KUKA KRL program: Wood_Test.src, Wood_Test.dat

--- Wood_Test.src ---
&ACCESS RVEO
&REL 9
&PARAM DISKPATH = KRC:\R1\Program\Milling
DEF Wood_Test ( )
   INT lnActSt,lnUsedBase,lnUsedTool,lnBaseNr
   INT lnJobNr, lncounter, lncounter2
   FRAME lfZcut
   FRAME lfToolDiamShift
   FRAME lfStartMillingPos
   FRAME lfBaseShift
   FRAME lfBaseCycleZ

   CONTINUE
   ;IF ($T1 OR $T2)THEN
   GLOBAL INTERRUPT DECL 3 WHEN $STOPMESS==TRUE DO IR_STOPM ( )
   INTERRUPT ON 3
   BAS (#INITMOV,0)
   lnActSt = 1
   PTP $POS_ACT
;;ptp xhome
   ;ENDIF

   ; PTP XHOME
   SpindleRun(grUsedRPM,#CLOCKWISE)

   PTP lAstartPos

   ; Used Base and tool
   lnUsedBase = 11
   lnUsedTool = 11

   gnLastToolNr = 4
   lnBaseNr = 21

   gfMillingOffset = $NULLFRAME


   lfZcut = $NULLFRAME
   lfZcut.Z = 0
   lfBaseShift = {X 0,Y 0,Z 0,A 0,B 0,C 0}
   lfBaseCycleZ = $NULLFRAME
   lfBaseCycleZ.Z = 0

   ;*************************************************************
   ;*                      Mill TOP SURFACE                     *
   ;*************************************************************
   lfBaseCycleZ = $NULLFRAME
   lfBaseCycleZ.Z = 0
   BASE_DATA[lnUsedBase] = BASE_DATA[lnBaseNr] : lfBaseShift : lfBaseCycleZ
   TOOL_DATA[lnUsedTool] = TOOL_DATA[gnLastToolNr] :{X 0,Y 0,Z 0,A 270,B 0,C 0}

   MoveSettings(lnUsedBase, lnUsedTool, 100, grUsedMillingSpeed)
   ;; Move To PreposMillingPos Point P5 {5mm far from WP surface}
   lfToolDiamShift   = $NULLFRAME
   lfToolDiamShift.X = 0
   lfToolDiamShift.Y = grTool_Diameter[4]
   lfToolDiamShift.Z = 5
   lfStartMillingPos = lfWorkPos[5] : lfToolDiamShift
   LIN lfStartMillingPos

   ;; Move To Milling Point P5
   MoveSettings(lnUsedBase, lnUsedTool, 100, grUsedMillingSpeed)
   lfToolDiamShift   =   $NULLFRAME
   lfToolDiamShift.x =  0
   lfToolDiamShift.Y =  grTool_Diameter[4]
   lfToolDiamShift.Z =  0
   LIN lfWorkPos[5]:lfToolDiamShift C_VEL

   ;; Move To Milling Point P6
   MoveSettings(lnUsedBase, lnUsedTool, 100, grUsedMillingSpeed)
   lfToolDiamShift   =   $NULLFRAME
   lfToolDiamShift.x =  0
   lfToolDiamShift.Y =  0;-grtool_diameter[4]
   lfToolDiamShift.Z =  0
   LIN lfWorkPos[6]:lfToolDiamShift C_VEL

   ;; Move To Milling Point P6
   MoveSettings(lnUsedBase, lnUsedTool, 100, grUsedMillingSpeed)
   lfToolDiamShift   =   $NULLFRAME
   lfToolDiamShift.x =  grtool_diameter[4] -10
   lfToolDiamShift.Y =  0;-grtool_diameter[4]
   lfToolDiamShift.Z =  0
   LIN lfWorkPos[6]:lfToolDiamShift C_VEL
    ;; Move To Milling Point P5
   MoveSettings(lnUsedBase, lnUsedTool, 100, grUsedMillingSpeed)
   lfToolDiamShift   =   $NULLFRAME
   lfToolDiamShift.x =  grTool_Diameter[4] -10
   lfToolDiamShift.Y =  grTool_Diameter[4]
   lfToolDiamShift.Z =  0
   LIN lfWorkPos[5]:lfToolDiamShift C_VEL

   MoveSettings(lnUsedBase, lnUsedTool, 100, 500)
   ;; End of Milling Move Out of the WP
   TRIGGER WHEN DISTANCE=1 DELAY=0 DO  SpindleSetSpeed(50) PRIO=-1
   LIN_REL {Z 5} C_VEL #TOOL

   LIN_REL {Z 100} C_VEL #BASE

   TOOL_DATA[lnUsedTool] = TOOL_DATA[gnLastToolNr] :{X 0,Y 0,Z 0,A 180,B 90,C -90}
   MoveSettings(lnUsedBase, lnUsedTool, 100, 500)
   PTP lastartpos C_PTP

END

--- Wood_Test.dat ---
&ACCESS RVEO
&REL 9
&PARAM DISKPATH = KRC:\R1\Program\Milling
DEFDAT  WOOD_TEST PUBLIC

DECL AXIS lAstartPos={A1 -14.2470465,A2 -67.0903091,A3 95.3724213,A4 83.6876450,A5 -70.3252869,A6 -65.7779922}
DECL FRAME lfPrePos[5]
lfPrePos[1]={X -32.0000,Y -50.0000,Z 350.000,A 90.0000,B 0.0,C -45.0000}
lfPrePos[2]={X -32.0000,Y -15.0000,Z 70.0000,A 90.0000,B 0.0,C -90.0000}
lfPrePos[3]={X 0.0,Y -32.0000,Z 70.0000,A 0.0,B 0.0,C 90.0000}
lfPrePos[4]={X 0.0,Y -32.0000,Z 50.0000,A 90.0000,B 0.0,C 0.0}
lfPrePos[5]={X 0.0,Y -50.0000,Z 350.000,A 90.0000,B 0.0,C 0.0}

DECL FRAME lfWorkPos[12]
lfWorkPos[1]={X 0.0,Y 0.0,Z 0.0,A 90.0000,B 0.0,C -90.0000}
lfWorkPos[2]={X 200.000,Y 0.0,Z 0.0,A 90.0000,B 0.0,C -90.0000}
lfWorkPos[3]={X 0.0,Y 0.0,Z 0.0,A 0.0,B 0.0,C 90.0000}
lfWorkPos[4]={X 0.0,Y 200.000,Z 0.0,A 0.0,B 0.0,C 90.0000}

lfWorkPos[5]={X 12.5000,Y 340.000,Z 0.0,A 0.0,B 0.0,C 0.0}
lfWorkPos[6]={X 12.5000,Y 12.5000,Z 0.0,A 0.0,B 0.0,C 0.0}
lfWorkPos[7]={X 200.000,Y 12.5000,Z 0.0,A 0.0,B 0.0,C 0.0}

lfWorkPos[8]={X 200.000,Y 1.00000,Z 0.0,A 0.0,B 0.0,C 45.0000}
lfWorkPos[9]={X 0.0,Y 1.00000,Z 0.0,A 0.0,B 0.0,C 45.0000}
lfWorkPos[10]={X 1.00000,Y 0.0,Z 0.0,A 0.0,B -45.0000,C 0.0}
lfWorkPos[11]={X 1.00000,Y 200.000,Z 0.0,A 0.0,B -45.0000,C 0.0}
ENDDAT
